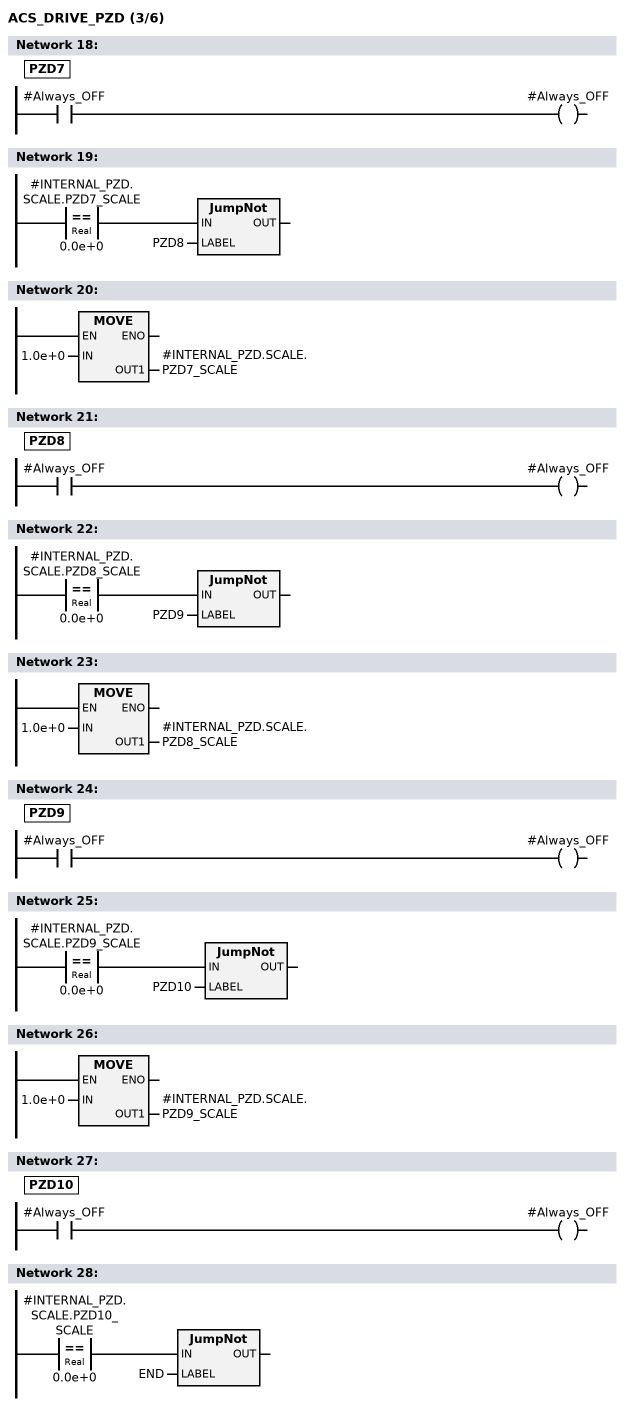
   Label( PZD7 )
   RUNG wire#powerrail
      Contact( #Always_OFF )
      Coil( #Always_OFF )
   END_RUNG
   // the same network as SCL:
   PZD7:
   #Always_OFF := #Always_OFF;
END_REGION

REGION Network 19
   // no SCL statement known for JumpNot: written as a call
   JumpNot(in := #INTERNAL_PZD.SCALE.PZD7_SCALE = 0.0e+0, label := PZD8);
END_REGION

REGION Network 20
   RUNG wire#powerrail
      { S7_GenerateENO := "TRUE" } Move(in := 1.0e+0, out1 => #INTERNAL_PZD.SCALE.PZD7_SCALE)
   END_RUNG
   // the same network as SCL:
   #INTERNAL_PZD.SCALE.PZD7_SCALE := 1.0e+0;
END_REGION

REGION Network 21
   Label( PZD8 )
   RUNG wire#powerrail
      Contact( #Always_OFF )
      Coil( #Always_OFF )
   END_RUNG
   // the same network as SCL:
   PZD8:
   #Always_OFF := #Always_OFF;
END_REGION

REGION Network 22
   // no SCL statement known for JumpNot: written as a call
   JumpNot(in := #INTERNAL_PZD.SCALE.PZD8_SCALE = 0.0e+0, label := PZD9);
END_REGION

REGION Network 23
   RUNG wire#powerrail
      { S7_GenerateENO := "TRUE" } Move(in := 1.0e+0, out1 => #INTERNAL_PZD.SCALE.PZD8_SCALE)
   END_RUNG
   // the same network as SCL:
   #INTERNAL_PZD.SCALE.PZD8_SCALE := 1.0e+0;
END_REGION

REGION Network 24
   Label( PZD9 )
   RUNG wire#powerrail
      Contact( #Always_OFF )
      Coil( #Always_OFF )
   END_RUNG
   // the same network as SCL:
   PZD9:
   #Always_OFF := #Always_OFF;
END_REGION

REGION Network 25
   // no SCL statement known for JumpNot: written as a call
   JumpNot(in := #INTERNAL_PZD.SCALE.PZD9_SCALE = 0.0e+0, label := PZD10);
END_REGION

REGION Network 26
   RUNG wire#powerrail
      { S7_GenerateENO := "TRUE" } Move(in := 1.0e+0, out1 => #INTERNAL_PZD.SCALE.PZD9_SCALE)
   END_RUNG
   // the same network as SCL:
   #INTERNAL_PZD.SCALE.PZD9_SCALE := 1.0e+0;
END_REGION

REGION Network 27
   Label( PZD10 )
   RUNG wire#powerrail
      Contact( #Always_OFF )
      Coil( #Always_OFF )
   END_RUNG
   // the same network as SCL:
   PZD10:
   #Always_OFF := #Always_OFF;
END_REGION

REGION Network 28
   // no SCL statement known for JumpNot: written as a call
   JumpNot(in := #INTERNAL_PZD.SCALE.PZD10_SCALE = 0.0e+0, label := END);
END_REGION

REGION Network 29
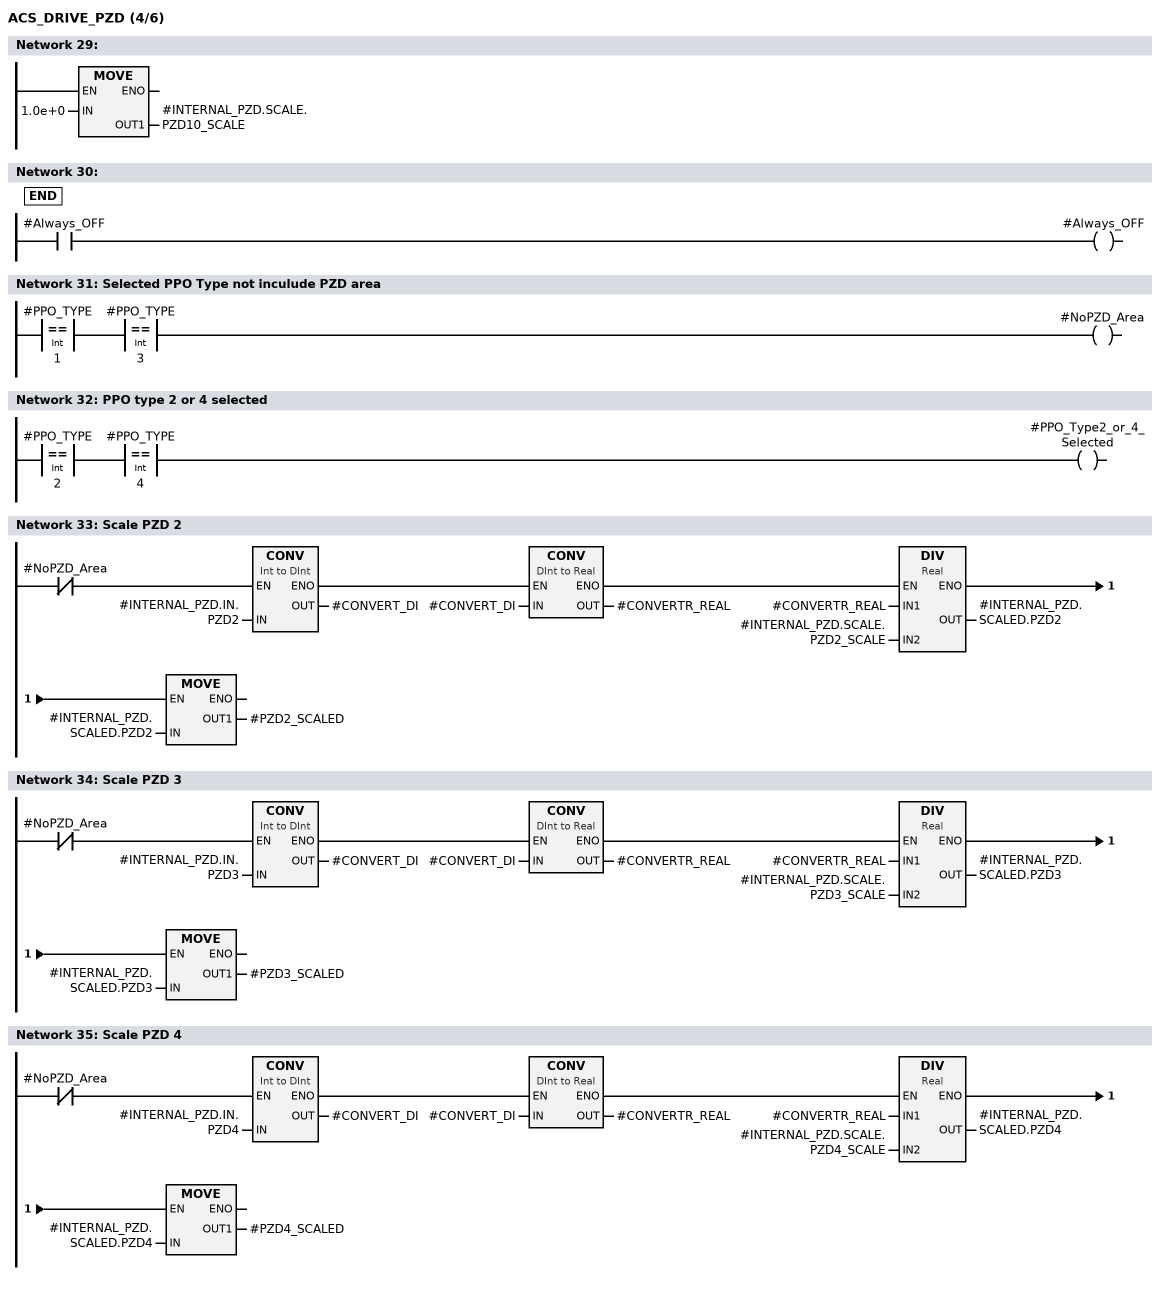
   RUNG wire#powerrail
      { S7_GenerateENO := "TRUE" } Move(in := 1.0e+0, out1 => #INTERNAL_PZD.SCALE.PZD10_SCALE)
   END_RUNG
   // the same network as SCL:
   #INTERNAL_PZD.SCALE.PZD10_SCALE := 1.0e+0;
END_REGION

REGION Network 30
   Label( END )
   RUNG wire#powerrail
      Contact( #Always_OFF )
      Coil( #Always_OFF )
   END_RUNG
   // the same network as SCL:
   END:
   #Always_OFF := #Always_OFF;
END_REGION

REGION Network 31: Selected PPO Type not inculude PZD area
   RUNG wire#powerrail
      { S7_Templates := "SrcType := Int" } EQ_Contact(in1 := #PPO_TYPE, in2 := 1)
      { S7_Templates := "SrcType := Int" } EQ_Contact(in1 := #PPO_TYPE, in2 := 3)
      Coil( #NoPZD_Area )
   END_RUNG
   // the same network as SCL:
   #NoPZD_Area := (#PPO_TYPE = 1) AND (#PPO_TYPE = 3);
END_REGION

REGION Network 32: PPO type 2 or 4 selected
   RUNG wire#powerrail
      { S7_Templates := "SrcType := Int" } EQ_Contact(in1 := #PPO_TYPE, in2 := 2)
      { S7_Templates := "SrcType := Int" } EQ_Contact(in1 := #PPO_TYPE, in2 := 4)
      Coil( #PPO_Type2_or_4_Selected )
   END_RUNG
   // the same network as SCL:
   #PPO_Type2_or_4_Selected := (#PPO_TYPE = 2) AND (#PPO_TYPE = 4);
END_REGION

REGION Network 33: Scale PZD 2
   RUNG wire#powerrail
      I_Contact( #NoPZD_Area )
      { S7_Templates := "[SrcType := Int, DestType := DInt]"; S7_GenerateENO := "TRUE" } Convert(in := #INTERNAL_PZD.IN.PZD2, out => #CONVERT_DI)
      { S7_Templates := "[SrcType := DInt, DestType := Real]"; S7_GenerateENO := "TRUE" } Convert(in := #CONVERT_DI, out => #CONVERTR_REAL)
      { S7_Templates := "SrcType := Real"; S7_GenerateENO := "TRUE" } Div(in1 := #CONVERTR_REAL, in2 := #INTERNAL_PZD.SCALE.PZD2_SCALE, out => #INTERNAL_PZD.SCALED.PZD2)
      { S7_GenerateENO := "TRUE" } Move(in := #INTERNAL_PZD.SCALED.PZD2, out1 => #PZD2_SCALED)
   END_RUNG
   // the same network as SCL:
   // ENO of a box is taken as its EN; it also drops when the box reports an error
   IF NOT #NoPZD_Area THEN
       #CONVERT_DI := INT_TO_DINT(#INTERNAL_PZD.IN.PZD2);
       #CONVERTR_REAL := DINT_TO_REAL(#CONVERT_DI);
       #INTERNAL_PZD.SCALED.PZD2 := #CONVERTR_REAL / #INTERNAL_PZD.SCALE.PZD2_SCALE;
       #PZD2_SCALED := #INTERNAL_PZD.SCALED.PZD2;
   END_IF;
END_REGION

REGION Network 34: Scale PZD 3
   RUNG wire#powerrail
      I_Contact( #NoPZD_Area )
      { S7_Templates := "[SrcType := Int, DestType := DInt]"; S7_GenerateENO := "TRUE" } Convert(in := #INTERNAL_PZD.IN.PZD3, out => #CONVERT_DI)
      { S7_Templates := "[SrcType := DInt, DestType := Real]"; S7_GenerateENO := "TRUE" } Convert(in := #CONVERT_DI, out => #CONVERTR_REAL)
      { S7_Templates := "SrcType := Real"; S7_GenerateENO := "TRUE" } Div(in1 := #CONVERTR_REAL, in2 := #INTERNAL_PZD.SCALE.PZD3_SCALE, out => #INTERNAL_PZD.SCALED.PZD3)
      { S7_GenerateENO := "TRUE" } Move(in := #INTERNAL_PZD.SCALED.PZD3, out1 => #PZD3_SCALED)
   END_RUNG
   // the same network as SCL:
   // ENO of a box is taken as its EN; it also drops when the box reports an error
   IF NOT #NoPZD_Area THEN
       #CONVERT_DI := INT_TO_DINT(#INTERNAL_PZD.IN.PZD3);
       #CONVERTR_REAL := DINT_TO_REAL(#CONVERT_DI);
       #INTERNAL_PZD.SCALED.PZD3 := #CONVERTR_REAL / #INTERNAL_PZD.SCALE.PZD3_SCALE;
       #PZD3_SCALED := #INTERNAL_PZD.SCALED.PZD3;
   END_IF;
END_REGION

REGION Network 35: Scale PZD 4
   RUNG wire#powerrail
      I_Contact( #NoPZD_Area )
      { S7_Templates := "[SrcType := Int, DestType := DInt]"; S7_GenerateENO := "TRUE" } Convert(in := #INTERNAL_PZD.IN.PZD4, out => #CONVERT_DI)
      { S7_Templates := "[SrcType := DInt, DestType := Real]"; S7_GenerateENO := "TRUE" } Convert(in := #CONVERT_DI, out => #CONVERTR_REAL)
      { S7_Templates := "SrcType := Real"; S7_GenerateENO := "TRUE" } Div(in1 := #CONVERTR_REAL, in2 := #INTERNAL_PZD.SCALE.PZD4_SCALE, out => #INTERNAL_PZD.SCALED.PZD4)
      { S7_GenerateENO := "TRUE" } Move(in := #INTERNAL_PZD.SCALED.PZD4, out1 => #PZD4_SCALED)
   END_RUNG
   // the same network as SCL:
   // ENO of a box is taken as its EN; it also drops when the box reports an error
   IF NOT #NoPZD_Area THEN
       #CONVERT_DI := INT_TO_DINT(#INTERNAL_PZD.IN.PZD4);
       #CONVERTR_REAL := DINT_TO_REAL(#CONVERT_DI);
       #INTERNAL_PZD.SCALED.PZD4 := #CONVERTR_REAL / #INTERNAL_PZD.SCALE.PZD4_SCALE;
       #PZD4_SCALED := #INTERNAL_PZD.SCALED.PZD4;
   END_IF;
END_REGION

REGION Network 36: Scale PZD 5
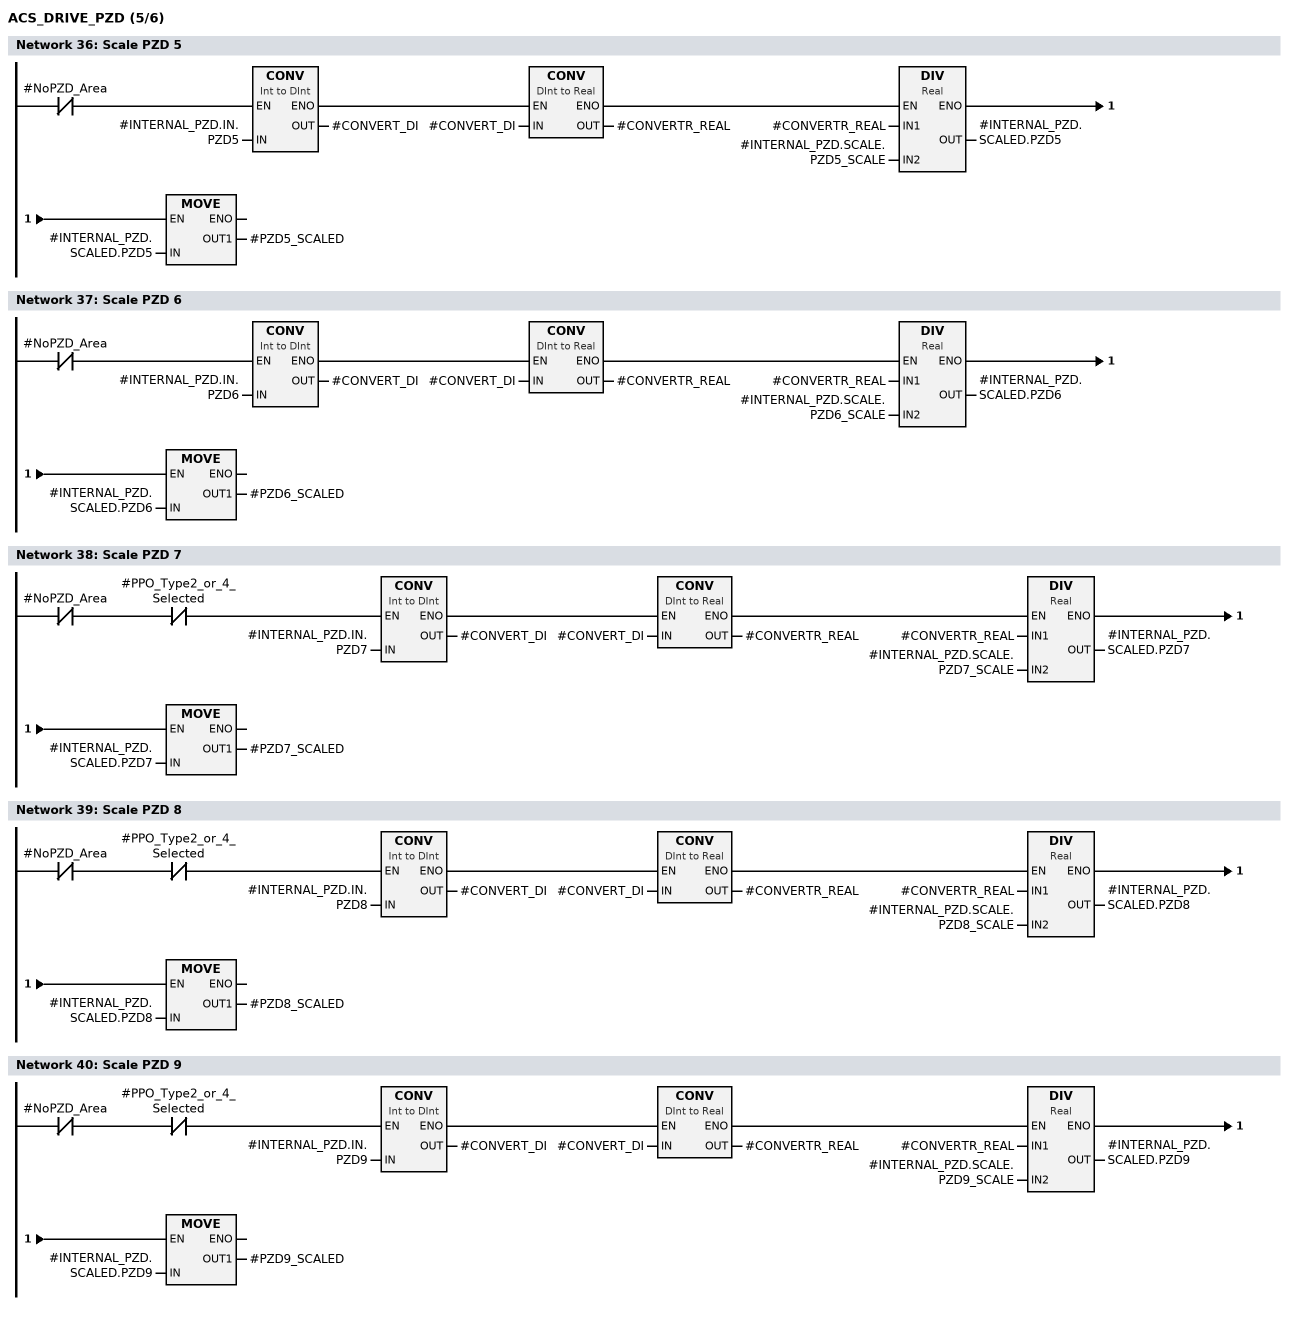
   RUNG wire#powerrail
      I_Contact( #NoPZD_Area )
      { S7_Templates := "[SrcType := Int, DestType := DInt]"; S7_GenerateENO := "TRUE" } Convert(in := #INTERNAL_PZD.IN.PZD5, out => #CONVERT_DI)
      { S7_Templates := "[SrcType := DInt, DestType := Real]"; S7_GenerateENO := "TRUE" } Convert(in := #CONVERT_DI, out => #CONVERTR_REAL)
      { S7_Templates := "SrcType := Real"; S7_GenerateENO := "TRUE" } Div(in1 := #CONVERTR_REAL, in2 := #INTERNAL_PZD.SCALE.PZD5_SCALE, out => #INTERNAL_PZD.SCALED.PZD5)
      { S7_GenerateENO := "TRUE" } Move(in := #INTERNAL_PZD.SCALED.PZD5, out1 => #PZD5_SCALED)
   END_RUNG
   // the same network as SCL:
   // ENO of a box is taken as its EN; it also drops when the box reports an error
   IF NOT #NoPZD_Area THEN
       #CONVERT_DI := INT_TO_DINT(#INTERNAL_PZD.IN.PZD5);
       #CONVERTR_REAL := DINT_TO_REAL(#CONVERT_DI);
       #INTERNAL_PZD.SCALED.PZD5 := #CONVERTR_REAL / #INTERNAL_PZD.SCALE.PZD5_SCALE;
       #PZD5_SCALED := #INTERNAL_PZD.SCALED.PZD5;
   END_IF;
END_REGION

REGION Network 37: Scale PZD 6
   RUNG wire#powerrail
      I_Contact( #NoPZD_Area )
      { S7_Templates := "[SrcType := Int, DestType := DInt]"; S7_GenerateENO := "TRUE" } Convert(in := #INTERNAL_PZD.IN.PZD6, out => #CONVERT_DI)
      { S7_Templates := "[SrcType := DInt, DestType := Real]"; S7_GenerateENO := "TRUE" } Convert(in := #CONVERT_DI, out => #CONVERTR_REAL)
      { S7_Templates := "SrcType := Real"; S7_GenerateENO := "TRUE" } Div(in1 := #CONVERTR_REAL, in2 := #INTERNAL_PZD.SCALE.PZD6_SCALE, out => #INTERNAL_PZD.SCALED.PZD6)
      { S7_GenerateENO := "TRUE" } Move(in := #INTERNAL_PZD.SCALED.PZD6, out1 => #PZD6_SCALED)
   END_RUNG
   // the same network as SCL:
   // ENO of a box is taken as its EN; it also drops when the box reports an error
   IF NOT #NoPZD_Area THEN
       #CONVERT_DI := INT_TO_DINT(#INTERNAL_PZD.IN.PZD6);
       #CONVERTR_REAL := DINT_TO_REAL(#CONVERT_DI);
       #INTERNAL_PZD.SCALED.PZD6 := #CONVERTR_REAL / #INTERNAL_PZD.SCALE.PZD6_SCALE;
       #PZD6_SCALED := #INTERNAL_PZD.SCALED.PZD6;
   END_IF;
END_REGION

REGION Network 38: Scale PZD 7
   RUNG wire#powerrail
      I_Contact( #NoPZD_Area )
      I_Contact( #PPO_Type2_or_4_Selected )
      { S7_Templates := "[SrcType := Int, DestType := DInt]"; S7_GenerateENO := "TRUE" } Convert(in := #INTERNAL_PZD.IN.PZD7, out => #CONVERT_DI)
      { S7_Templates := "[SrcType := DInt, DestType := Real]"; S7_GenerateENO := "TRUE" } Convert(in := #CONVERT_DI, out => #CONVERTR_REAL)
      { S7_Templates := "SrcType := Real"; S7_GenerateENO := "TRUE" } Div(in1 := #CONVERTR_REAL, in2 := #INTERNAL_PZD.SCALE.PZD7_SCALE, out => #INTERNAL_PZD.SCALED.PZD7)
      { S7_GenerateENO := "TRUE" } Move(in := #INTERNAL_PZD.SCALED.PZD7, out1 => #PZD7_SCALED)
   END_RUNG
   // the same network as SCL:
   // ENO of a box is taken as its EN; it also drops when the box reports an error
   IF NOT #NoPZD_Area AND NOT #PPO_Type2_or_4_Selected THEN
       #CONVERT_DI := INT_TO_DINT(#INTERNAL_PZD.IN.PZD7);
       #CONVERTR_REAL := DINT_TO_REAL(#CONVERT_DI);
       #INTERNAL_PZD.SCALED.PZD7 := #CONVERTR_REAL / #INTERNAL_PZD.SCALE.PZD7_SCALE;
       #PZD7_SCALED := #INTERNAL_PZD.SCALED.PZD7;
   END_IF;
END_REGION

REGION Network 39: Scale PZD 8
   RUNG wire#powerrail
      I_Contact( #NoPZD_Area )
      I_Contact( #PPO_Type2_or_4_Selected )
      { S7_Templates := "[SrcType := Int, DestType := DInt]"; S7_GenerateENO := "TRUE" } Convert(in := #INTERNAL_PZD.IN.PZD8, out => #CONVERT_DI)
      { S7_Templates := "[SrcType := DInt, DestType := Real]"; S7_GenerateENO := "TRUE" } Convert(in := #CONVERT_DI, out => #CONVERTR_REAL)
      { S7_Templates := "SrcType := Real"; S7_GenerateENO := "TRUE" } Div(in1 := #CONVERTR_REAL, in2 := #INTERNAL_PZD.SCALE.PZD8_SCALE, out => #INTERNAL_PZD.SCALED.PZD8)
      { S7_GenerateENO := "TRUE" } Move(in := #INTERNAL_PZD.SCALED.PZD8, out1 => #PZD8_SCALED)
   END_RUNG
   // the same network as SCL:
   // ENO of a box is taken as its EN; it also drops when the box reports an error
   IF NOT #NoPZD_Area AND NOT #PPO_Type2_or_4_Selected THEN
       #CONVERT_DI := INT_TO_DINT(#INTERNAL_PZD.IN.PZD8);
       #CONVERTR_REAL := DINT_TO_REAL(#CONVERT_DI);
       #INTERNAL_PZD.SCALED.PZD8 := #CONVERTR_REAL / #INTERNAL_PZD.SCALE.PZD8_SCALE;
       #PZD8_SCALED := #INTERNAL_PZD.SCALED.PZD8;
   END_IF;
END_REGION

REGION Network 40: Scale PZD 9
   RUNG wire#powerrail
      I_Contact( #NoPZD_Area )
      I_Contact( #PPO_Type2_or_4_Selected )
      { S7_Templates := "[SrcType := Int, DestType := DInt]"; S7_GenerateENO := "TRUE" } Convert(in := #INTERNAL_PZD.IN.PZD9, out => #CONVERT_DI)
      { S7_Templates := "[SrcType := DInt, DestType := Real]"; S7_GenerateENO := "TRUE" } Convert(in := #CONVERT_DI, out => #CONVERTR_REAL)
      { S7_Templates := "SrcType := Real"; S7_GenerateENO := "TRUE" } Div(in1 := #CONVERTR_REAL, in2 := #INTERNAL_PZD.SCALE.PZD9_SCALE, out => #INTERNAL_PZD.SCALED.PZD9)
      { S7_GenerateENO := "TRUE" } Move(in := #INTERNAL_PZD.SCALED.PZD9, out1 => #PZD9_SCALED)
   END_RUNG
   // the same network as SCL:
   // ENO of a box is taken as its EN; it also drops when the box reports an error
   IF NOT #NoPZD_Area AND NOT #PPO_Type2_or_4_Selected THEN
       #CONVERT_DI := INT_TO_DINT(#INTERNAL_PZD.IN.PZD9);
       #CONVERTR_REAL := DINT_TO_REAL(#CONVERT_DI);
       #INTERNAL_PZD.SCALED.PZD9 := #CONVERTR_REAL / #INTERNAL_PZD.SCALE.PZD9_SCALE;
       #PZD9_SCALED := #INTERNAL_PZD.SCALED.PZD9;
   END_IF;
END_REGION

REGION Network 41: Scale PZD 10
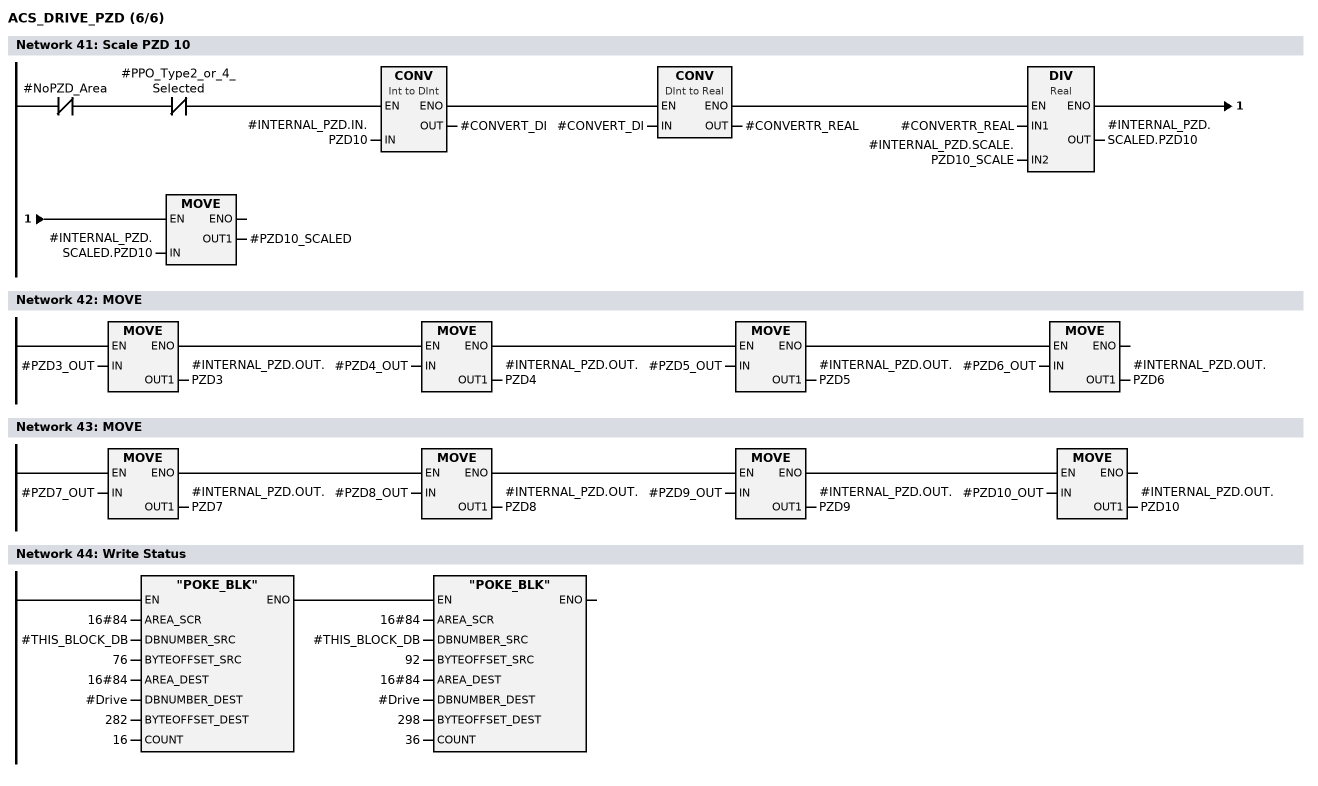
   RUNG wire#powerrail
      I_Contact( #NoPZD_Area )
      I_Contact( #PPO_Type2_or_4_Selected )
      { S7_Templates := "[SrcType := Int, DestType := DInt]"; S7_GenerateENO := "TRUE" } Convert(in := #INTERNAL_PZD.IN.PZD10, out => #CONVERT_DI)
      { S7_Templates := "[SrcType := DInt, DestType := Real]"; S7_GenerateENO := "TRUE" } Convert(in := #CONVERT_DI, out => #CONVERTR_REAL)
      { S7_Templates := "SrcType := Real"; S7_GenerateENO := "TRUE" } Div(in1 := #CONVERTR_REAL, in2 := #INTERNAL_PZD.SCALE.PZD10_SCALE, out => #INTERNAL_PZD.SCALED.PZD10)
      { S7_GenerateENO := "TRUE" } Move(in := #INTERNAL_PZD.SCALED.PZD10, out1 => #PZD10_SCALED)
   END_RUNG
   // the same network as SCL:
   // ENO of a box is taken as its EN; it also drops when the box reports an error
   IF NOT #NoPZD_Area AND NOT #PPO_Type2_or_4_Selected THEN
       #CONVERT_DI := INT_TO_DINT(#INTERNAL_PZD.IN.PZD10);
       #CONVERTR_REAL := DINT_TO_REAL(#CONVERT_DI);
       #INTERNAL_PZD.SCALED.PZD10 := #CONVERTR_REAL / #INTERNAL_PZD.SCALE.PZD10_SCALE;
       #PZD10_SCALED := #INTERNAL_PZD.SCALED.PZD10;
   END_IF;
END_REGION

REGION Network 42: MOVE
   RUNG wire#powerrail
      { S7_GenerateENO := "TRUE" } Move(in := #PZD3_OUT, out1 => #INTERNAL_PZD.OUT.PZD3)
      { S7_GenerateENO := "TRUE" } Move(in := #PZD4_OUT, out1 => #INTERNAL_PZD.OUT.PZD4)
      { S7_GenerateENO := "TRUE" } Move(in := #PZD5_OUT, out1 => #INTERNAL_PZD.OUT.PZD5)
      { S7_GenerateENO := "TRUE" } Move(in := #PZD6_OUT, out1 => #INTERNAL_PZD.OUT.PZD6)
   END_RUNG
   // the same network as SCL:
   // ENO of a box is taken as its EN; it also drops when the box reports an error
   #INTERNAL_PZD.OUT.PZD3 := #PZD3_OUT;
   #INTERNAL_PZD.OUT.PZD4 := #PZD4_OUT;
   #INTERNAL_PZD.OUT.PZD5 := #PZD5_OUT;
   #INTERNAL_PZD.OUT.PZD6 := #PZD6_OUT;
END_REGION

REGION Network 43: MOVE
   RUNG wire#powerrail
      { S7_GenerateENO := "TRUE" } Move(in := #PZD7_OUT, out1 => #INTERNAL_PZD.OUT.PZD7)
      { S7_GenerateENO := "TRUE" } Move(in := #PZD8_OUT, out1 => #INTERNAL_PZD.OUT.PZD8)
      { S7_GenerateENO := "TRUE" } Move(in := #PZD9_OUT, out1 => #INTERNAL_PZD.OUT.PZD9)
      { S7_GenerateENO := "TRUE" } Move(in := #PZD10_OUT, out1 => #INTERNAL_PZD.OUT.PZD10)
   END_RUNG
   // the same network as SCL:
   // ENO of a box is taken as its EN; it also drops when the box reports an error
   #INTERNAL_PZD.OUT.PZD7 := #PZD7_OUT;
   #INTERNAL_PZD.OUT.PZD8 := #PZD8_OUT;
   #INTERNAL_PZD.OUT.PZD9 := #PZD9_OUT;
   #INTERNAL_PZD.OUT.PZD10 := #PZD10_OUT;
END_REGION

REGION Network 44: Write Status
   RUNG wire#powerrail
      "POKE_BLK"(AREA_SCR := 16#84, DBNUMBER_SRC := #THIS_BLOCK_DB, BYTEOFFSET_SRC := 76, AREA_DEST := 16#84, DBNUMBER_DEST := #Drive, BYTEOFFSET_DEST := 282, COUNT := 16)
      "POKE_BLK"(AREA_SCR := 16#84, DBNUMBER_SRC := #THIS_BLOCK_DB, BYTEOFFSET_SRC := 92, AREA_DEST := 16#84, DBNUMBER_DEST := #Drive, BYTEOFFSET_DEST := 298, COUNT := 36)
   END_RUNG
   // the same network as SCL:
   "POKE_BLK"(AREA_SCR := 16#84,
              DBNUMBER_SRC := #THIS_BLOCK_DB,
              BYTEOFFSET_SRC := 76,
              AREA_DEST := 16#84,
              DBNUMBER_DEST := #Drive,
              BYTEOFFSET_DEST := 282,
              COUNT := 16,
              ENO => #_w1);
   IF #_w1 THEN
       "POKE_BLK"(AREA_SCR := 16#84,
                  DBNUMBER_SRC := #THIS_BLOCK_DB,
                  BYTEOFFSET_SRC := 92,
                  AREA_DEST := 16#84,
                  DBNUMBER_DEST := #Drive,
                  BYTEOFFSET_DEST := 298,
                  COUNT := 36);
   END_IF;
END_REGION
END_FUNCTION_BLOCK

FUNCTION "POKE" : Void   // FC1, SCL
TITLE = POKE Block
{ S7_Optimized_Access := 'TRUE' }
AUTHOR : ABB
FAMILY : DRIVES
NAME : ABB
VERSION : 1.2
   VAR_INPUT
      DB_Number : DB_ANY;
      byteOffset : DInt;
      Input_Value : DInt;
   END_VAR
BEGIN
   POKE(area := 16#84,
        dbNumber := #DB_Number,
        byteOffset := #byteOffset,
        value := #Input_Value);
END_FUNCTION

FUNCTION "POKE_BLK" : Void   // FC2, SCL
TITLE = POKE_BLK
{ S7_Optimized_Access := 'TRUE' }
AUTHOR : ABB
FAMILY : DRIVES
NAME : ABB
VERSION : 1.2
   VAR_INPUT
      AREA_SCR : Byte;
      DBNUMBER_SRC : DB_ANY;
      BYTEOFFSET_SRC : DInt;
      AREA_DEST : Byte;
      DBNUMBER_DEST : DB_ANY;
      BYTEOFFSET_DEST : DInt;
      COUNT : DInt;
   END_VAR
BEGIN
   POKE_BLK(area_src := #AREA_SCR,
            dbNumber_src := #DBNUMBER_SRC,
            byteOffset_src := #BYTEOFFSET_SRC,
            area_dest := #AREA_DEST,
            dbNumber_dest := #DBNUMBER_DEST,
            byteOffset_dest := #BYTEOFFSET_DEST,
            count := #COUNT);
END_FUNCTION